VAR_GLOBAL CONSTANT
    TcUnit_ResultExportXmlPath : T_MaxString :=
        'C:\TwinCAT\3.1\Boot\Plc\TcUnitResults.xml';
END_VAR

(* stored: Version 1.1.0.1
   GVL GVL_TcUnit: Id {9f6a422a-b3f5-424c-993f-d5e89d7da1f6} *)
